Universal Robots PolyScope program: future_is_now.urp

Program future_is_now (installation=default directory=/home/ur/ursim-current/programs createdIn=5.11.5.1010327 lastSavedIn=5.11.8.1010444 robotSerialNumber=20195599999)
Calibrated DH parameters: a=[0, -0.425, -0.3922, 0, 0, 0]; d=[0.1625, 0, 0, 0.1333, 0.0997, 0.0996]; alpha=[1.570796, 0, 0, 1.570796, -1.570796, 0]; deltaTheta=[0, 0, 0, 0, 0, 0]
InitVariablesNode variables(variable(name=poseReady, expression=False), variable(name=rx, expression=1.171), variable(name=ry, expression=1.171), variable(name=rz, expression=1.233), variable(name=x, expression=-0.098), variable(name=y, expression=0.133), variable(name=z, expression=0.695))
Robot Program (runOnlyOnce=false)
  poseReady := read_input_boolean_register(64)
  x := read_input_float_register(0)
  y := read_input_float_register(1)
  z := read_input_float_register(2)
  rx := read_input_float_register(3)
  ry := read_input_float_register(4)
  rz := read_input_float_register(5)
  If poseReady
    rotation := rpy2rotvec([rx,ry,rz])
    q := get_inverse_kin(p[x, y, z, rotation[0], rotation[1],rotation[2]])
    Script: servoj(q, lookahead_time=0.2, gain=100)
  Else 
    Script: movej([-3.14,-2.89,1.91,-2.21,4.71,3.14],a=1.2,v=0.3,t=0,r=0)
